PROGRAM PRG_FaultHandling
VAR
	
	i							: INT;
	bFlagResetOn				: BOOL;
	bStationCycleFaultFlag		: BOOL;




END_VAR
VAR_IN_OUT

  aAlarms  : ARRAY[0..2] OF ST_Events;
END_VAR

ACT_FaultTrig();

(************************************** Faults reset **********************************************)
IF   GVL_HMI_GLOBAL.bResetButton THEN 
	FOR i := 0 TO 127 DO
		GVL_MASTER.stAlarms[0].aEventFlags[i] := FALSE;
	END_FOR
END_IF


//===============================================================
//Initialize event texts on first scan
IF NOT GVL_MASTER.stAlarms[0].bEventTextsSet THEN
	SetEventTexts();
	GVL_MASTER.stAlarms[0].bEventTextsSet := TRUE;
END_IF
IF NOT GVL_MASTER.stAlarms[0].bEventTextsSet THEN
	GVL_MASTER.stAlarms[0].bEventTextsSet := FALSE;
END_IF


(***************************************************************************************************)
//Immediate fault
GVL_MASTER.stAlarms[0].bImmediateFault := FALSE;
FOR i := 0 TO 32DO
	GVL_MASTER.stAlarms[0].bImmediateFault := GVL_MASTER.stAlarms[0].bImmediateFault OR GVL_MASTER.stAlarms[0].aEventFlags[i];
END_FOR

//Cycle stop fault
GVL_MASTER.stAlarms[0].bCycleStopFault := FALSE;
FOR i := 33 TO 79 DO
	GVL_MASTER.stAlarms[0].bCycleStopFault := GVL_MASTER.stAlarms[0].bCycleStopFault OR GVL_MASTER.stAlarms[0].aEventFlags[i];
END_FOR

//Cycle stop request
GVL_MASTER.stAlarms[0].bCycleStopRequest := FALSE;
FOR i := 80 TO 99 DO
	GVL_MASTER.stAlarms[0].bCycleStopRequest := GVL_MASTER.stAlarms[0].bCycleStopRequest OR GVL_MASTER.stAlarms[0].aEventFlags[i];
END_FOR


(**************************** Master Fault Monitors ***********************************************)
(* Station Immediate Fault Monitor *)
GVL_MASTER.stMasterControl.bNoStationImmediateFault := 	NOT GVL_MASTER.stAlarms[0].bImmediateFault AND NOT GVL_MASTER.stAlarms[1].bImmediateFault AND
                                            			NOT GVL_MASTER.stAlarms[2].bImmediateFault;

(**************************************************************************************************)
(**************************** Cycle stop falt  **************************************)
bStationCycleFaultFlag := NOT GVL_MASTER.stAlarms[0].bCycleStopFault AND NOT GVL_MASTER.stAlarms[1].bCycleStopFault AND
                          NOT GVL_MASTER.stAlarms[2].bCycleStopFault;

(**************************** Master Immediate Fault Monitor **************************************)
GVL_MASTER.stMasterControl.bNoMachineImmediateFault := NOT GVL_MASTER.stAlarms[0].bImmediateFault AND NOT GVL_MASTER.stAlarms[1].bImmediateFault AND
                                            NOT GVL_MASTER.stAlarms[2].bImmediateFault;

									
(**************************************************************************************************)

(* Master Cycle Stop Fault Monitor *)
GVL_MASTER.stMasterControl.bNoCycleStopFault := NOT GVL_MASTER.stAlarms[0].bCycleStopFault;

ACTION ACT_FaultTrig:
(**************************************************************************************************)
(**************************** Master Immediate Fault Stop *****************************************)
(**************************************************************************************************)

//Beckhoff EL1809 Not Operational
IF NOT GVL_MASTER.stMachineStatus.bSystemPowerUp AND GVL_IO.dwTerminalInfo[3].nTerminal_State<>8 THEN
	GVL_MASTER.stAlarms[0].aEventFlags[33] := TRUE;
END_IF
//Beckhoff EL2809 Not Operational
IF NOT GVL_MASTER.stMachineStatus.bSystemPowerUp AND GVL_IO.dwTerminalInfo[4].nTerminal_State<>8 THEN
	GVL_MASTER.stAlarms[0].aEventFlags[34] := TRUE;
END_IF
//System stopping timeout
GVL_MASTER.stAlarms[0].aEventTimers[38](IN := ( GVL_MASTER.stMachineStatus.bSystemStopping ), PT := T#20S);
IF GVL_MASTER.stAlarms[0].aEventTimers[38].Q THEN
	GVL_MASTER.stAlarms[0].aEventFlags[38] := TRUE;	
END_IF
//User not Log In
GVL_MASTER.stAlarms[0].aEventTimers[39](IN := (NOT GVL_HMI_GLOBAL.bUserLogedIntSignal), PT := T#40MS);
IF GVL_MASTER.stAlarms[0].aEventTimers[39].Q THEN
	GVL_MASTER.stAlarms[0].aEventFlags[39] := TRUE;	
END_IF
//User LOG-Off Timeout Manual Mode
GVL_MASTER.stAlarms[0].aEventTimers[40](IN:= ((NOT GVL_HMI_GLOBAL.bUserLogedIntSignal) AND GVL_MASTER.stMachineStatus.bManualMode),PT:= T#1S); 
IF GVL_MASTER.stAlarms[0].aEventTimers[40].Q THEN
	GVL_MASTER.stAlarms[0].aEventFlags[40] := TRUE;
END_IF
//Keyence DL-P1 Error
IF GVL_IO.dw_B08_DL_PN1.dldErrorStt THEN
	GVL_MASTER.stAlarms[0].aEventFlags[41] := TRUE;
END_IF
//10 Min Auto cycle stop
IF PRG_MasterCycle.bAutoCycleStop  THEN //
	GVL_MASTER.stAlarms[0].aEventFlags[80] := TRUE;
END_IF
//Autocyle Timeout 
GVL_MASTER.stAlarms[0].aEventTimers[42](IN:= GVL_MASTER.stStationSruct[0].bStationInProgress, PT :=T#10M ); 
IF GVL_MASTER.stAlarms[0].aEventTimers[42].Q THEN
	GVL_MASTER.stAlarms[0].aEventFlags[42] := TRUE;
END_IF
//Part removed during process WHEN THE CLAMP IS ALLREADY DOWN o1
IF GVL_Master.stStationSruct[0].nState > 1000 AND GVL_Master.stStationSruct[0].nState < 2000 AND GVL_IO.dw_T02_EL1809.iCalmpClosed AND NOT GVL_IO.dw_T02_EL1809.iPartPresent THEN
	GVL_MASTER.stAlarms[0].aEventFlags[43] := TRUE;
END_IF

//Clamp toggled before requested
IF GVL_Master.stStationSruct[0].nState > 1132 AND GVL_Master.stStationSruct[0].nState < 1700 AND NOT GVL_IO.dw_T02_EL1809.iCalmpClosed THEN
	GVL_MASTER.stAlarms[0].aEventFlags[45] := TRUE;
END_IF
//Press Acknowledge
IF GVL_HMI_GLOBAL.bAutocycleFaultDialog THEN
	GVL_MASTER.stAlarms[0].aEventFlags[46] := TRUE;
END_IF

//Remove Nest **LA 18092025
IF GVL_HMI_GLOBAL.bStartButton AND NOT PRG_Mastercycle.biClamp AND PRG_Mastercycle.biPartPresent THEN 
	GVL_MASTER.stAlarms[0].aEventFlags[100] := TRUE;
	ELSIF NOT PRG_Mastercycle.biPartPresent THEN 
		GVL_MASTER.stAlarms[0].aEventFlags[100] := FALSE;
END_IF

//Release Clamp  **LA 18092025
IF GVL_HMI_GLOBAL.bStartButton AND PRG_Mastercycle.biClamp AND NOT PRG_Mastercycle.biPartPresent AND GVL_MASTER.stMachineStatus.bSystemReadyToStart THEN 
	GVL_MASTER.stAlarms[0].aEventFlags[101] := TRUE;
	ELSIF NOT PRG_Mastercycle.biClamp THEN 
		GVL_MASTER.stAlarms[0].aEventFlags[101] := FALSE;
END_IF

//Releas Clamp and Remove Nest  **LA 18092025
IF GVL_HMI_GLOBAL.bStartButton AND PRG_Mastercycle.biClamp AND PRG_Mastercycle.biPartPresent AND GVL_MASTER.stMachineStatus.bSystemReadyToStart THEN
	GVL_MASTER.stAlarms[0].aEventFlags[102] := TRUE;
	ELSIF  NOT PRG_Mastercycle.biClamp AND NOT PRG_Mastercycle.biPartPresent THEN
		GVL_MASTER.stAlarms[0].aEventFlags[102] := FALSE;
END_IF
END_ACTION

METHOD PRIVATE SetEventTexts : BOOL
VAR_INPUT
END_VAR
//Immediate Faults
GVL_MASTER.stAlarms[0].aEventTexts[0] := 'SPARE';
GVL_MASTER.stAlarms[0].aEventTexts[1] := 'SPARE';
GVL_MASTER.stAlarms[0].aEventTexts[2] := 'SPARE';
GVL_MASTER.stAlarms[0].aEventTexts[3] := 'SPARE';
GVL_MASTER.stAlarms[0].aEventTexts[4] := '';
GVL_MASTER.stAlarms[0].aEventTexts[5] := '';
GVL_MASTER.stAlarms[0].aEventTexts[6] := '';
GVL_MASTER.stAlarms[0].aEventTexts[7] := '';
GVL_MASTER.stAlarms[0].aEventTexts[8] := '';
GVL_MASTER.stAlarms[0].aEventTexts[9] := '';
GVL_MASTER.stAlarms[0].aEventTexts[10] := '';
GVL_MASTER.stAlarms[0].aEventTexts[10] := ''; 
GVL_MASTER.stAlarms[0].aEventTexts[11] := '';
GVL_MASTER.stAlarms[0].aEventTexts[12] := '';
GVL_MASTER.stAlarms[0].aEventTexts[13] := '';
GVL_MASTER.stAlarms[0].aEventTexts[14] := '';
GVL_MASTER.stAlarms[0].aEventTexts[15] := '';


//Cycle stop fault

GVL_MASTER.stAlarms[0].aEventTexts[33] := 'Beckhoff EL1809 Not Operational';
GVL_MASTER.stAlarms[0].aEventTexts[34] := 'Beckhoff EL2809 Not Operational';
GVL_MASTER.stAlarms[0].aEventTexts[35] := '';
GVL_MASTER.stAlarms[0].aEventTexts[36] := '';
GVL_MASTER.stAlarms[0].aEventTexts[37] := '';
GVL_MASTER.stAlarms[0].aEventTexts[38] := 'Master - Stopping timeout';
GVL_MASTER.stAlarms[0].aEventTexts[39] := 'User Not Log IN';
GVL_MASTER.stAlarms[0].aEventTexts[40] := 'User Log-Off Timeout Manual Mode'; 
GVL_MASTER.stAlarms[0].aEventTexts[41] := 'Keyence DL-P1 Error';
GVL_MASTER.stAlarms[0].aEventTexts[42] := 'Autocyle Timeou' ;
GVL_MASTER.stAlarms[0].aEventTexts[43] := 'Part removed during cycle';
GVL_MASTER.stAlarms[0].aEventTexts[44] := 'Clamp toggled before requested';
GVL_MASTER.stAlarms[0].aEventTexts[45] := 'Clamp toggled before requested';
GVL_MASTER.stAlarms[0].aEventTexts[46] := 'Press Acknowledge';
GVL_MASTER.stAlarms[0].aEventTexts[47] := '';
GVL_MASTER.stAlarms[0].aEventTexts[48] := '';
GVL_MASTER.stAlarms[0].aEventTexts[59] := '';
GVL_MASTER.stAlarms[0].aEventTexts[50] := '';

//Cycle Stop Requests

GVL_MASTER.stAlarms[0].aEventTexts[80] := 'Machine Cycle Stop 10 Min Not Use Timeout';
GVL_MASTER.stAlarms[0].aEventTexts[81] := '';
GVL_MASTER.stAlarms[0].aEventTexts[82] := '';

GVL_MASTER.stAlarms[0].aEventTexts[84] := '';
GVL_MASTER.stAlarms[0].aEventTexts[85] := '';
GVL_MASTER.stAlarms[0].aEventTexts[86] := '';
GVL_MASTER.stAlarms[0].aEventTexts[87] := ''; 
GVL_MASTER.stAlarms[0].aEventTexts[88] := '';
GVL_MASTER.stAlarms[0].aEventTexts[89] := '';

// Message //**LA 18092025
GVL_MASTER.stAlarms[0].aEventTexts[100] := 'Remove Nest';
GVL_MASTER.stAlarms[0].aEventTexts[101] := 'Release Clamp';
GVL_MASTER.stAlarms[0].aEventTexts[102] := 'Release Clamp and Remove Nest';
END_METHOD

END_PROGRAM

(* stored: Version 1.1.0.1, ProductVersion 3.1.4024.13
   POU PRG_FaultHandling: Id {1ed57a34-1c0a-4c7e-a0fc-90a123d0d2dc}, SpecialFunc None
   Action ACT_FaultTrig: Id {f82952b9-10cd-47a6-a8aa-cbbe9096c605}
   Method SetEventTexts: Id {84625549-67f8-41bf-b81a-cc5fcd6308ae} *)
